KUKA KRL data list: Signals.dat

&ACCESS RV
DEFDAT SIGNALS PUBLIC
ENDDAT
